(* CoDeSys 2.3 export: ST_PumpConfig.exp *)

(* Data type in Pump *)
(* єЮЭдШУгаРжШп ЭРбЮбР *)
TYPE ST_PumpConfig :
STRUCT
    (* ЅЮЬШЭРЫмЭлХ ЯРаРЬХвал ЭРбЮбР *)
    rNominalFlow : REAL := 100.0;          (* Ь?/з *)
    rNominalHead : REAL := 50.0;           (* Ь *)
    rNominalPower : REAL := 15.0;          (* ЪІв *)
    rNominalCurrent : REAL := 30.0;        (* ° *)
    rNominalSpeed : REAL := 2950.0;        (* ЮС/ЬШЭ *)
    
    (* АРСЮзШХ ФШРЯРЧЮЭл *)
    rMinFlow : REAL := 10.0;               (* Ь?/з *)
    rMaxFlow : REAL := 120.0;              (* Ь?/з *)
    rMinInletPressure : REAL := 0.5;       (* СРа *)
    rMaxOutletPressure : REAL := 10.0;     (* СРа *)
    rMinFrequency : REAL := 20.0;          (* іж *)
    rMaxFrequency : REAL := 50.0;          (* іж *)
    
    (* ГбвРТЪШ ЧРйШв *)
    rDryRunFlowLimit : REAL := 5.0;        (* Ь?/з *)
    rClosedValveFlowLimit : REAL := 2.0;   (* Ь?/з *)
    rCavitationNPSH : REAL := 3.0;         (* Ь *)
    rOverloadCurrentLimit : REAL := 110.0;  (* % Юв ЭЮЬШЭРЫР *)
    rLowEfficiencyLimit : REAL := 60.0;    (* % *)
    
    (* ВРЩЬХал ЧРйШв *)
    tDryRunDelay : TIME := T#10S;
    tClosedValveDelay : TIME := T#30S;
    tCavitationDelay : TIME := T#5S;
    tOverloadDelay : TIME := T#10S;
    tStartupTime : TIME := T#20S;
    tStopTime : TIME := T#10S;
    
    (* НЪбЯЫгРвРжШЮЭЭлХ ЯРаРЬХвал *)
    iMaxStartsPerHour : INT := 6;          (* јРЪб ЯгбЪЮТ Т зРб *)
END_STRUCT
END_TYPE
